Staubli VAL3: chkLife.pgx

public program chkLife()
  local num l_i
  local string l_sMsg
begin
  //检查IO连接是否正常
  blifebit_all_ok=true
  for l_i=0 to nAxesSum-1
    if ioStatus(diReady2SwOn[l_i])<0
      blifebit[l_i]=false
      l_sMsg="第"+toString("",l_i+1)+"轴通讯异常"
      popUpMsg(l_sMsg)
      logMsg(l_sMsg)
      blifebit_all_ok=blifebit_all_ok and blifebit[l_i]
      return
    else
      blifebit[l_i]=true
      blifebit_all_ok=blifebit_all_ok and blifebit[l_i]
    endIf
  endFor

end
